// TwinCAT 3 PLC project Untitled1
// ProgramVersion: 3.1.4024.0
// libraries:
//   Tc2_Standard, * (Beckhoff Automation GmbH)
//   Tc2_System, * (Beckhoff Automation GmbH)
//   Tc3_Module, * (Beckhoff Automation GmbH)
// project tree:
//   FB/ FB_AppelEtage.TcPOU
//   / Gestionnaire de visualisation.TcVMO (not stored), GlobalTextList.TcGTLO, PlcTask.TcTTO
//   GVLs/ GVL.TcGVL
//   POUs/ MAIN.TcPOU
//   VISUs/ Visualization.TcVIS

CONFIGURATION Untitled1
    RESOURCE PLC ON TwinCAT3
        TASK PlcTask(INTERVAL := T#10ms, PRIORITY := 20);
        PROGRAM MAIN WITH PlcTask : MAIN;
    END_RESOURCE
END_CONFIGURATION

// ---- GVLs/GVL.TcGVL
{attribute 'qualified_only'}
VAR_GLOBAL
	// Bouton appelle ascenseur etage
	BP_EG : BOOL := FALSE;
	BP_1OG : BOOL := FALSE;
	BP_2OG : BOOL := FALSE;
	
	// Lampe 
	Lampe_EG : BOOL := FALSE;
	Lampe_1OG : BOOL := FALSE;
	Lampe_2OG : BOOL := FALSE;
	
	iEtageAppel : INT;
	iEtageActuel : INT; 
	
	MouvementAscenseur : BOOL := FALSE;
	TempsMouvementAscenseur : TON;
	
	// Ouverture Porte
	OuverturePorte : Ton;
	Lampe_Ouverture : BOOL := FALSE;
	
	// Fermeture Porte
	FermeturePorte : Ton;
	Lampe_Fermeture : Bool := False;
	
END_VAR

// ---- POUs/MAIN.TcPOU
PROGRAM MAIN
VAR
    rTrig_BP_EG  : R_TRIG;
    rTrig_BP_1OG : R_TRIG;
    rTrig_BP_2OG : R_TRIG;
END_VAR

rTrig_BP_EG(CLK := GVL.BP_EG);
rTrig_BP_1OG(CLK := GVL.BP_1OG);
rTrig_BP_2OG(CLK := GVL.BP_2OG);

// Appelle bouton etage
IF rTrig_BP_EG.Q THEN
	GVL.iEtageAppel := 0;
	gvl.MouvementAscenseur := TRUE;
END_IF

IF rTrig_BP_1OG.Q THEN
	GVL.iEtageAppel := 1;
	gvl.MouvementAscenseur := TRUE;
END_IF

IF rTrig_BP_2OG.Q THEN
	GVL.iEtageAppel := 2;
	gvl.MouvementAscenseur := TRUE;
END_IF

// Fermeture porte
IF gvl.MouvementAscenseur THEN
	gvl.FermeturePorte (In := TRUE, PT :=  T#5S);
END_IF

// Durée du trajet
IF gvl.FermeturePorte.Q THEN
	
	// Lampe Fermeture
	gvl.Lampe_Fermeture := TRUE;	
	gvl.Lampe_Ouverture := False;

	// Lampe témoin chaque étage
	gvl.Lampe_EG := FALSE;
	gvl.Lampe_1OG := FALSE;
	gvl.Lampe_2OG := false;
	
	// Calcul du temps
	CASE ABS(GVL.iEtageAppel - GVL.iEtageActuel) OF

        0: GVL.TempsMouvementAscenseur (IN := TRUE, PT := T#0S);
        1: GVL.TempsMouvementAscenseur (IN := TRUE, PT := T#5S);
        2: GVL.TempsMouvementAscenseur (IN := TRUE, PT := T#10S);
		
    END_CASE
	
	// Arrivé a l'étage demandé
	IF GVL.TempsMouvementAscenseur.Q THEN
        GVL.iEtageActuel := GVL.iEtageAppel;
        gvl.MouvementAscenseur := FALSE;
        GVL.TempsMouvementAscenseur(IN := FALSE);
		
		CASE GVL.iEtageActuel OF
			0:
				GVL.BP_EG := FALSE;
				GVL.Lampe_EG := TRUE;
		
			1:
				GVL.BP_1OG := FALSE;
				GVL.Lampe_1OG := TRUE;
		
			2:
				GVL.BP_2OG := FALSE;
				GVL.Lampe_2OG := TRUE;
		END_CASE
		
		gvl.Lampe_Fermeture := FALSE;
		
		// Ouverture porte
		gvl.OuverturePorte (In := TRUE, PT :=  T#5S);
		
		IF gvl.OuverturePorte.Q THEN
			gvl.Lampe_Ouverture := TRUE;
		END_IF
    END_IF
END_IF

END_PROGRAM

// ---- FB/FB_AppelEtage.TcPOU
FUNCTION_BLOCK FB_AppelEtage

VAR_INPUT
	
END_VAR

VAR_OUTPUT
	
END_VAR

VAR
	
END_VAR

END_FUNCTION_BLOCK

// ---- GlobalTextList.TcGTLO
TEXTLIST GlobalTextList
  853 = '1 OG'
  506 = '2 OG'
  44 = 'EG'
  698 = 'Fermeture'
  260 = 'Ouverture'
  657 = 'RDC'
END_TEXTLIST

// ---- VISUs/Visualization.TcVIS
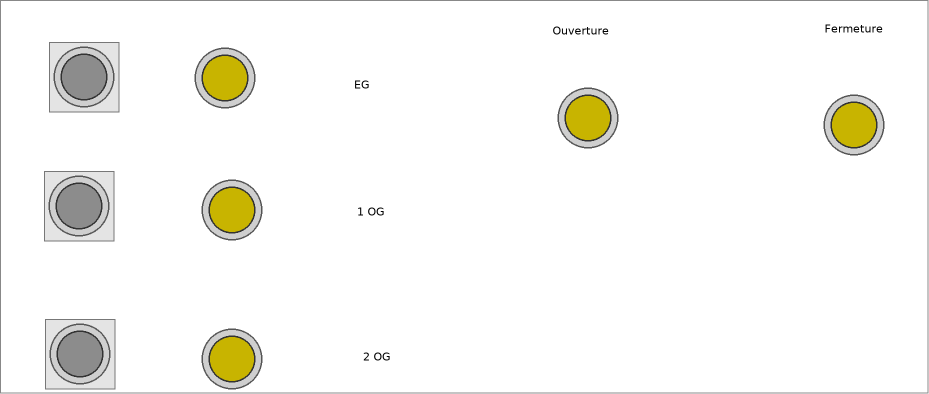
VISUALIZATION Visualization  // 929x394
    PushSwitch (49,42 70x70), variable: GVL.BP_EG, behaviour: TOGGLE, style: Switch-PushSwitch-Gray
    PushSwitch (44,171 70x70), variable: GVL.BP_1OG, behaviour: TOGGLE, style: Switch-PushSwitch-Gray
    PushSwitch (45,319 70x70), variable: GVL.BP_2OG, behaviour: TOGGLE, style: Switch-PushSwitch-Gray
    Label (287,70 150x30), "EG"
    Label (296,197 150x30), "1 OG"
    Label (302,342 150x30), "2 OG"
    Lamp1 (190,43 70x70), variable: GVL.Lampe_EG, style: Lamp-Lamp1-Yellow
    Lamp1 (197,175 70x70), variable: GVL.Lampe_1OG, style: Lamp-Lamp1-Yellow
    Lamp1 (197,324 70x70), variable: GVL.Lampe_2OG, style: Lamp-Lamp1-Yellow
    Lamp1 (553,83 70x70), variable: GVL.Lampe_Ouverture, style: Lamp-Lamp1-Yellow
    Lamp1 (819,90 70x70), variable: GVL.Lampe_Fermeture, style: Lamp-Lamp1-Yellow
    Label (506,16 150x30), "Ouverture"
    Label (779,14 150x30), "Fermeture"
END_VISUALIZATION
